// Mitsubishi GX Works2 project: 240416_지연간격동작회로   PLC: Q03UDV

PROGRAM MAIN
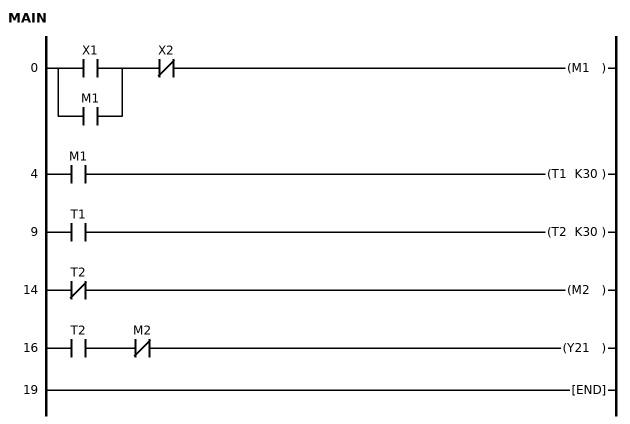
0     LD      X1
      OR      M1
      ANI     X2
      OUT     M1
4     LD      M1
      OUT     T1 K30
9     LD      T1
      OUT     T2 K30
14    LDI     T2
      OUT     M2
16    LD      T2
      ANI     M2
      OUT     Y21
19    END
END_PROGRAM
